Fanuc KAREL source: kb00196.KL

-- PROVISIONAL review KL for V1013-1; original PC SHA256 5a1e170aa821813912d2c54d1543be80616d5113d937424104aef07dabe19c42
-- Incomplete behavior may be omitted. Consult companion uncertainty JSON. Do not deploy.
PROGRAM KB00196
%NOLOCKGROUP
BEGIN
  -- UNRESOLVED_PC offsets 5-14; opcodes 3F,75
  -- UNRESOLVED_PC offsets 19-26; opcodes 9D,23
  -- UNRESOLVED_PC offsets 31-38; opcodes 9D,23
  -- UNRESOLVED_PC offsets 43-52; opcodes 3F,75
  -- UNRESOLVED_PC offsets 57-89; opcodes 27,22,2A,22,22,22,2A,31
  -- UNRESOLVED_PC offsets 94-98; opcodes 7F
END KB00196
